FUNCTION_BLOCK "LAF_GetSinaEpos"
TITLE = LAF_GetSinaEpos
{ S7_Optimized_Access := 'TRUE' ; Published := 'TRUE' }
AUTHOR : 'Siemens Digital Industries'
FAMILY : LAF
VERSION : 1.2
//This block reads EPOS positioning status information as well as setpoint and actual values from a SINAMICS drive via acyclic communication depending on the configured type of SINAMICS and the selected drive object index in the HMI by the operator.
   VAR_INPUT
      enable { S7_PredefinedAssignment := 'TRUE'} : Bool := TRUE;   // FALSE = Disables functionality of FB from user program (optional), FB is normally enabled via HMI ('moduleInterface.hmi.sinaEposScreenActive' = TRUE)
   END_VAR

   VAR_OUTPUT
      valid { ExternalWritable := 'False'} : Bool;   // Valid set of output values available at the FB
      busy { ExternalWritable := 'False'} : Bool;   // FB is not finished and new output values can be expected
      error { ExternalWritable := 'False'} : Bool;   // An error occurred during the execution of the FB, for details see diagnostics output
      status { ExternalWritable := 'False'} : Word := #STATUS_NO_CALL;   // 16#0000 - 16#7FFF: Status of the FB, 16#8000 - 16#FFFF: Error identification
      diagnostics { ExternalWritable := 'False'} : "LAF_typeDiagnostics";   // Diagnostics information of FB
      statusWriteRecord { ExternalAccessible := 'False'; ExternalVisible := 'False'; ExternalWritable := 'False'} : DWord;   // Status output of WRREC
      statusReadRecord { ExternalAccessible := 'False'; ExternalVisible := 'False'; ExternalWritable := 'False'} : DWord;   // Status output of RDREC
   END_VAR

   VAR_IN_OUT
      configuration { S7_PredefinedAssignment := 'DriveDiagConfig.driveObjects'} : Array[*] of "LAF_typeDriveDiagConfig";
      moduleInterface { S7_PredefinedAssignment := 'DriveDiagInterfaceHmi.diagStatus'} : "LAF_typeDriveDiagInterfaceHmi";
   END_VAR

   VAR
      statInternal { ExternalAccessible := 'False'; ExternalVisible := 'False'; ExternalWritable := 'False'} : Struct   // Static structure for internal tags
         enablePrevious { ExternalAccessible := 'False'; ExternalVisible := 'False'; ExternalWritable := 'False'} : Bool;   // Previous value of 'enable' input for edge detection
         valid { ExternalAccessible := 'False'; ExternalVisible := 'False'; ExternalWritable := 'False'} : Bool;   // Value for output 'valid'
         busy { ExternalAccessible := 'False'; ExternalVisible := 'False'; ExternalWritable := 'False'} : Bool;   // Value for output 'busy'
         error { ExternalAccessible := 'False'; ExternalVisible := 'False'; ExternalWritable := 'False'} : Bool;   // Value for output 'error'
         errorUserCleared { ExternalAccessible := 'False'; ExternalVisible := 'False'; ExternalWritable := 'False'} : Bool;   // Error occurred that can only be solved by user; rising edge at enable input necessary
         errorAutoCleared { ExternalAccessible := 'False'; ExternalVisible := 'False'; ExternalWritable := 'False'} : Bool;   // Error occurred that can be acknowledged by FB
         disablingCompleted { ExternalAccessible := 'False'; ExternalVisible := 'False'; ExternalWritable := 'False'} : Bool;   // TRUE: Disabling has been completed
         diagnostics { ExternalAccessible := 'False'; ExternalVisible := 'False'; ExternalWritable := 'False'; S7_SetPoint := 'False'} : "LAF_typeDiagnostics" := (#STATUS_NO_CALL, (), ());
         emptyDiagnostics { ExternalAccessible := 'False'; ExternalVisible := 'False'; ExternalWritable := 'False'; S7_SetPoint := 'False'} : "LAF_typeDiagnostics" := (#STATUS_NO_CALL, (), ());   // Empty diagnostics information (for initialization purposes only)
      END_STRUCT;
      statMainState { ExternalAccessible := 'False'; ExternalVisible := 'False'; ExternalWritable := 'False'} : DInt := #FB_STATE_NO_PROCESSING;   // State in the state machine of the FB
      statArrayMin { ExternalAccessible := 'False'; ExternalVisible := 'False'; ExternalWritable := 'False'} : DInt;   // Lower bound of configuration array
      statArrayMax { ExternalAccessible := 'False'; ExternalVisible := 'False'; ExternalWritable := 'False'} : DInt;   // Upper bound of configuration array
      instWriteRecord {InstructionName := 'WRREC'; LibVersion := '1.1'; ExternalAccessible := 'False'; ExternalVisible := 'False'; ExternalWritable := 'False'; S7_SetPoint := 'False'} : WRREC;   // Instance of WRREC
      instReadRecord {InstructionName := 'RDREC'; LibVersion := '1.0'; ExternalAccessible := 'False'; ExternalVisible := 'False'; ExternalWritable := 'False'; S7_SetPoint := 'False'} : RDREC;   // Instance of RDREC
      statWriteReq { ExternalAccessible := 'False'; ExternalVisible := 'False'; ExternalWritable := 'False'} : Struct   // Data of write record according to parameter request
         header { ExternalAccessible := 'False'; ExternalVisible := 'False'; ExternalWritable := 'False'} : Struct   // Request header
            reqRef { ExternalAccessible := 'False'; ExternalVisible := 'False'; ExternalWritable := 'False'} : Byte;   // Unique identification of the request/response pair for the IO controller. The IO device mirrors the request reference in its response
            reqID { ExternalAccessible := 'False'; ExternalVisible := 'False'; ExternalWritable := 'False'} : Byte;   // Specifies the type of request (0x01=read, 0x02=write)
            axis { ExternalAccessible := 'False'; ExternalVisible := 'False'; ExternalWritable := 'False'} : Byte := 16#01;   // Specifies the drive object number for a drive unit with more than one drive object
            noPara { ExternalAccessible := 'False'; ExternalVisible := 'False'; ExternalWritable := 'False'} : Byte := 16#01;   // Number of parameters
         END_STRUCT;
         data { ExternalAccessible := 'False'; ExternalVisible := 'False'; ExternalWritable := 'False'} : Array[0..#DATA_ARRY_MAX] of Byte;   // Request data
      END_STRUCT;
      statReadReq { ExternalAccessible := 'False'; ExternalVisible := 'False'; ExternalWritable := 'False'} : Struct   // Data of read record according to parameter response
         header { ExternalAccessible := 'False'; ExternalVisible := 'False'; ExternalWritable := 'False'} : Struct   // Request header
            reqRef { ExternalAccessible := 'False'; ExternalVisible := 'False'; ExternalWritable := 'False'} : Byte;   // Mirrowed request reference in response of the IO device.
            reqID { ExternalAccessible := 'False'; ExternalVisible := 'False'; ExternalWritable := 'False'} : Byte;   // Mirrowed request identifier. Specifies if request execution was positive or negative (0x01=read+, 0x02=write+, 0x81=read-, 0x82=write-)
            axis { ExternalAccessible := 'False'; ExternalVisible := 'False'; ExternalWritable := 'False'} : Byte := 16#01;   // Specifies the drive object number for a drive unit with more than one drive object
            noPara { ExternalAccessible := 'False'; ExternalVisible := 'False'; ExternalWritable := 'False'} : Byte := 16#01;   // Number of parameters
         END_STRUCT;
         data { ExternalAccessible := 'False'; ExternalVisible := 'False'; ExternalWritable := 'False'} : Array[0..#DATA_ARRY_MAX] of Byte;   // Request data
      END_STRUCT;
      instActTimer {InstructionName := 'IEC_TIMER'; LibVersion := '1.0'; ExternalAccessible := 'False'; ExternalVisible := 'False'; ExternalWritable := 'False'; S7_SetPoint := 'False'} : IEC_TIMER;   // Instance of actual timer for
      instReqTimer {InstructionName := 'IEC_TIMER'; LibVersion := '1.0'; ExternalAccessible := 'False'; ExternalVisible := 'False'; ExternalWritable := 'False'; S7_SetPoint := 'False'} : IEC_TIMER;   // Instance of request timer to retrigger write request
      statDataTransRun { ExternalAccessible := 'False'; ExternalVisible := 'False'; ExternalWritable := 'False'} : Bool;   // Data transfer is running
      statWriteReqSet { ExternalAccessible := 'False'; ExternalVisible := 'False'; ExternalWritable := 'False'} : Bool;   // Parameter for write request set
      statActTimerIn { ExternalAccessible := 'False'; ExternalVisible := 'False'; ExternalWritable := 'False'} : Bool;   // Actual timer start input
      statPrevTimeValue { ExternalAccessible := 'False'; ExternalVisible := 'False'; ExternalWritable := 'False'} : Time;   // Timer value of last trigger
      statActTimerValueAct { ExternalAccessible := 'False'; ExternalVisible := 'False'; ExternalWritable := 'False'} : Time;   // Current timer value of actual timer
      statActTimerValueReq { ExternalAccessible := 'False'; ExternalVisible := 'False'; ExternalWritable := 'False'} : Time;   // Current timer value of request timer
      statPrevDriveIndex { ExternalAccessible := 'False'; ExternalVisible := 'False'; ExternalWritable := 'False'} : DInt;   // Previous drive index
   END_VAR

   VAR_TEMP
      tempEnable : Bool;   // Temporary value for input 'enable'
      tempReferenceDesignator : WString[128];   // Temporary value for inout 'referenceDesignator'
      tempDriveIndex : DInt;   // Temporary value for inout 'driveIndex'
      tempSinaType : UInt;   // Temporary value for inout 'sinaType'
      tempSinaHwID : HW_IO;   // Temporary value for inout 'sinaHwID'
      tempDriveObjectNo : USInt;   // Temporary value for inout 'driveObjectNo'
      tempActTimerOut : Bool;   // Actual timer output
      tempReadReqTimerOut : Bool;   // Request timer output
      tempValueWord : Word;   // Temporary value for 16bit
      tempValueDword : DWord;   // Temporary value for 32bit
   END_VAR

   VAR CONSTANT
      FB_STATE_NO_PROCESSING : DInt := 0;   // FB state: No processing
      FB_STATE_ENABLING : DInt := 10;   // FB state: Enabling
      FB_STATE_PROCESSING : DInt := 50;   // FB state: Processing
      FB_STATE_DISABLING : DInt := 90;   // FB state: Disabling
      STATUS_NO_CALL : Word := 16#7000;   // No job being currently processed
      STATUS_FIRST_CALL : Word := 16#7001;   // First call after incoming new job (rising edge 'enable')
      STATUS_SUBSEQUENT_CALL : Word := 16#7002;   // Subsequent call during active processing without further details
      STATUS_WARN_ARRY_MIN : Word := 16#7003;   // Active processing with index assigned to lower bound of configuration arry
      STATUS_WARN_ARRY_MAX : Word := 16#7004;   // Active processing with index assigned to upper bound of configuration arry
      STAUTS_WARN_NO_SINAMICS : Word := 16#7005;   // Selected SINAMICS type in configuration not supported. Active processing with SINAMICS type assigned to no type.
      STAUTS_WARN_DO_SINGLE_AXIS : Word := 16#7006;   // Active processing with drive object number assigned to single-axis
      SUB_STATUS_NO_ERROR : Word := 16#0000;   // NO error occurred in sub function call
      ERR_UNDEFINED_STATE : Word := 16#8600;   // Error: due to an undefined state in state machine
      DIM_ARRAY_CONFIG : UDInt := 1;   // Dimension of the configuration array
      DRV_INDEX_INIT : DInt := -1;   // Initial value for drive index
      DRV_DO_SINGLE_AXIS : USInt := 1;   // Drive object number for single-axis
      DATA_ARRY_MAX : UInt := 235;   // Maximum size in bytes for request/response data
      DPV1_INDEX_DB47 : DInt := 47;   // DPV1 services PROFIBUS/PROFINET: Data block 47
      DPV1_LENGH_DATA : UInt := 240;   // DPV1 services PROFIBUS/PROFINET: Maximum length in bytes of the data record information
      TYPE_OF_SINA_NO_TYPE : UInt := 0;   // Type of SINAMICS not specified
      TYPE_OF_SINA_G120 : UInt := 114;   // Type of SINAMICS is G120
      TYPE_OF_SINA_G220 : UInt := 214;   // Type of SINAMICS is G220
      TYPE_OF_SINA_S120 : UInt := 124;   // Type of SINAMICS is S120
      TYPE_OF_SINA_S120_EPOS : UInt := 125;   // Type of SINAMICS is S120 with EPOS
      TYPE_OF_SINA_S200 : UInt := 220;   // Type of SINAMICS is S200
      TYPE_OF_SINA_S200_EPOS : UInt := 221;   // Type of SINAMICS is S200 with EPOS
      TYPE_OF_SINA_S210 : UInt := 222;   // Type of SINAMICS is S210
      TYPE_OF_SINA_S210_EPOS : UInt := 223;   // Type of SINAMICS is S210 with EPOS
      TYPE_OF_SINA_S220 : UInt := 224;   // Type of SINAMICS is S220
      TYPE_OF_SINA_S220_EPOS : UInt := 225;   // Type of SINAMICS is S220 with EPOS
      REQ_ID_READ : Byte := 16#01;   // Specifies read request for WRREC
      REQ_ID_WRITE : Byte := 16#02;   // Specifies write request for WRREC
      REQ_REF_G120 : Byte := 32;   // Response ID of response request of G120
      REQ_REF_G220 : Byte := 132;   // Response ID of response request of G220
      REQ_REF_S120 : Byte := 62;   // Response ID of response request of S120
      REQ_REF_S200 : Byte := 142;   // Response ID of response request of S200
      REQ_REF_S210 : Byte := 152;   // Response ID of response request of S210
      REQ_REF_S220 : Byte := 162;   // Response ID of response request of S220
   END_VAR


BEGIN
	REGION BLOCK INFO HEADER
	    //===============================================================================
	    // Siemens AG / (c)Copyright 2024
	    //-------------------------------------------------------------------------------
	    // Title:            LAF_GetSinaEpos
	    // Comment/Function: This block reads EPOS positioning status information as well
	    //                   as setpoint and actual values from a SINAMICS drive via
	    //                   acyclic communication depending on the configured type of
	    //                   SINAMICS and the selected drive object index in the HMI
	    //                   by the operator.
	    // Library/Family:   Automation Framework / Drive Diagnostic
	    // Author:           Siemens Digital Industries
	    // Tested with:      S7-PLCSIM Advanced 6.0
	    // Engineering:      TIA Portal V19
	    // Restrictions:     -
	    // Requirements:     -
	    //-------------------------------------------------------------------------------
	    // Change log table:
	    // Version  | Date       | Expert in charge        | Changes applied
	    //----------|------------|-------------------------|-----------------------------
	    // 01.00.00 | 15.12.2023 | SIMATIC Systems Support | First released version
	    // 01.01.00 | 30.06.2024 | SIMATIC Systems Support | UDTs updated, Enable/Disable
	    // 01.02.00 | 30.09.2024 | SIMATIC Systems Support | Block information properties updated
	    //===============================================================================
	END_REGION BLOCK INFO HEADER

	REGION DESCRIPTION
	(/*
	This block reads EPOS positioning status information as well as setpoint and actual values
	via PROFIBUS/PROFINET from a SINAMICS drive, by using acyclic communication with
	"Write data record" and "Read data record" services via the PROFIdrive parameter channel
	with data block 47 and the WRREC and RDREC system blocks.
	At runtime, this block is enabled when the SINAMCIS EPOS status diagnostic screen is shown
	in the HMI. Based on the selected drive object (index) in the HMI by the operator, the EPOS status
	is read out from the SINAMICS and transmitted to the HMI.
	The shown EPOS status in the HMI depends on the type of SINAMICS(S120_EPOS, S200_EPOS, S210_EPOS).
	Therefore the type of SINAMICS must be specified in the configuration DB. In addition, the
	hardware identifier (HW_IO) and the number of the drive object (DO) must be configured too.
	*/)
	END_REGION

	REGION INPUTS
	    // Work with temporary values / create process image
	    #tempEnable := #enable AND #moduleInterface.hmi.sinaEposScreenActive;
	    #tempDriveIndex := #moduleInterface.hmi.driveIndex;
	END_REGION INPUTS

	REGION ENABLING/DISABLING
	    IF (#tempEnable = TRUE) AND (#statInternal.diagnostics.status = #STATUS_NO_CALL) THEN // Enable FB
	        // First call; initialize FB
	        #statInternal.valid := TRUE;
	        #statInternal.busy := TRUE;
	        #statInternal.error := FALSE;
	        #statInternal.errorUserCleared := FALSE;
	        #statInternal.errorAutoCleared := FALSE;
	        #statInternal.disablingCompleted := FALSE;
	        #statInternal.diagnostics := #statInternal.emptyDiagnostics;
	        #diagnostics := #statInternal.emptyDiagnostics;
	        #statInternal.diagnostics.status := #STATUS_FIRST_CALL;
	        // State machine - start processing
	        #statMainState := #FB_STATE_ENABLING;
	        // Initialize diagnostic data
	        #statusWriteRecord := W#16#00;
	        #statusReadRecord := W#16#00;
	        #statPrevDriveIndex := #DRV_INDEX_INIT;
	        #moduleInterface.sina.sinaType := 0;
	        #moduleInterface.sina.statusWord := W#16#0;
	        #moduleInterface.sina.eposStatusWord1 := W#16#0;
	        #moduleInterface.sina.eposStatusWord2 := W#16#0;
	        #moduleInterface.sina.operatingDisplay := 0;
	        #moduleInterface.sina.override := 0.0;
	        #moduleInterface.sina.posSetValue := 0.0;
	        #moduleInterface.sina.posActValue := 0.0;
	        #moduleInterface.sina.velSetValue := 0.0;
	        #moduleInterface.sina.velActValue := 0.0;
	        #moduleInterface.sina.lengthUnit := 0;
	        #moduleInterface.sina.velocityUnit := 0;
	        #moduleInterface.sina.residualDistance := 0.0;
	        #moduleInterface.sina.followingError := 0.0;
	        #moduleInterface.sina.posControlWord := W#16#0;
	        #moduleInterface.sina.posStatusWord := W#16#0;
	        #moduleInterface.sina.blockSelected := 0;
	        #moduleInterface.sina.blockActive := 0;
	        #moduleInterface.sina.mdiPosSetValue := 0.0;

	    ELSIF (#tempEnable = FALSE) AND (#statInternal.enablePrevious = TRUE) THEN // Disable FB
	        #statMainState := #FB_STATE_DISABLING;

	    ELSIF (#statInternal.diagnostics.status = #STATUS_FIRST_CALL) THEN // Set status identifier of subsequent call
	        #statInternal.diagnostics.status := #STATUS_SUBSEQUENT_CALL;
	    END_IF;

	    // Edge detection 'tempEnable'
	    #statInternal.enablePrevious := #tempEnable;
	END_REGION ENABLING/DISABLING

	IF (#statInternal.diagnostics.status = #STATUS_NO_CALL) THEN // Nothing to do -> End here to reduce "system load"
	    RETURN;
	END_IF;

	REGION STATE MACHINE
	    CASE #statMainState OF // State machine of FB
	        #FB_STATE_NO_PROCESSING:
	            REGION No Processing
	                ; // No processing active (Note: this state must always be present and left empty)
	            END_REGION No Processing

	        #FB_STATE_ENABLING: // Enabling active
	            REGION Enabling
	                // Initialize boundaries of configuration array
	                #statArrayMin := LOWER_BOUND(ARR := #configuration, DIM := #DIM_ARRAY_CONFIG);
	                #statArrayMax := UPPER_BOUND(ARR := #configuration, DIM := #DIM_ARRAY_CONFIG);
	                // Continue processing with next state
	                #statMainState := #FB_STATE_PROCESSING;
	            END_REGION Enabling

	        #FB_STATE_PROCESSING: // Processing active
	            REGION Processing
	                // When index is off boundaries, index is assigned to violated bound and active processing with warning
	                IF (#tempDriveIndex < #statArrayMin) THEN
	                    #tempDriveIndex := #statArrayMin;
	                    #statInternal.diagnostics.status := #STATUS_WARN_ARRY_MIN;
	                    #statInternal.diagnostics.subfunctionStatus := #SUB_STATUS_NO_ERROR;
	                    #statInternal.diagnostics.stateNumber := #statMainState;
	                ELSIF (#tempDriveIndex > #statArrayMax) THEN
	                    #tempDriveIndex := #statArrayMax;
	                    #statInternal.diagnostics.status := #STATUS_WARN_ARRY_MAX;
	                    #statInternal.diagnostics.subfunctionStatus := #SUB_STATUS_NO_ERROR;
	                    #statInternal.diagnostics.stateNumber := #statMainState;
	                ELSE
	                    #statInternal.diagnostics.status := #STATUS_SUBSEQUENT_CALL;
	                    #statInternal.diagnostics.subfunctionStatus := #SUB_STATUS_NO_ERROR;
	                    #statInternal.diagnostics.stateNumber := #statMainState;
	                END_IF;

	                // Work with temporary values
	                #tempReferenceDesignator := #configuration[#tempDriveIndex].referenceDesignator;
	                #tempSinaType := #configuration[#tempDriveIndex].sinaType;
	                #tempSinaHwID := #configuration[#tempDriveIndex].sinaHwID;
	                #tempDriveObjectNo := #configuration[#tempDriveIndex].sinaDriveObjectNo;

	                // When SINAMICS type is not supported, type is assigned to no type
	                IF (#tempSinaType <> #TYPE_OF_SINA_G120) AND
	                    (#tempSinaType <> #TYPE_OF_SINA_S120) AND
	                    (#tempSinaType <> #TYPE_OF_SINA_S120_EPOS) AND
	                    (#tempSinaType <> #TYPE_OF_SINA_S200) AND
	                    (#tempSinaType <> #TYPE_OF_SINA_S200_EPOS) AND
	                    (#tempSinaType <> #TYPE_OF_SINA_S210) AND
	                    (#tempSinaType <> #TYPE_OF_SINA_S210_EPOS)
	                THEN
	                    #tempSinaType := #TYPE_OF_SINA_NO_TYPE;
	                    #statInternal.diagnostics.status := #STAUTS_WARN_NO_SINAMICS;
	                    #statInternal.diagnostics.subfunctionStatus := #SUB_STATUS_NO_ERROR;
	                    #statInternal.diagnostics.stateNumber := #statMainState;
	                END_IF;

	                // Check drive object number
	                IF (#tempDriveObjectNo < #DRV_DO_SINGLE_AXIS) THEN
	                    #tempDriveObjectNo := #DRV_DO_SINGLE_AXIS;
	                    #statInternal.diagnostics.status := #STAUTS_WARN_DO_SINGLE_AXIS;
	                    #statInternal.diagnostics.subfunctionStatus := #SUB_STATUS_NO_ERROR;
	                    #statInternal.diagnostics.stateNumber := #statMainState;
	                END_IF;

	                // Set SINAMICS type
	                #moduleInterface.sina.sinaType := #tempSinaType;

	                // Actual timer for communication with drive
	                #instActTimer.TON(IN := #statActTimerIn,
	                                  PT := T#596h,
	                                  Q => #tempActTimerOut,
	                                  ET => #statActTimerValueAct);
	                IF NOT #tempActTimerOut THEN
	                    #statActTimerIn := true;
	                ELSE
	                    #statActTimerIn := FALSE;
	                    #statPrevTimeValue := T#0s;
	                END_IF;

	                // Initialize dataö
	                IF #tempDriveIndex <> #statPrevDriveIndex THEN
	                    // Write request
	                    #statWriteReq.header.reqRef := B#16#00;
	                    #statWriteReq.header.reqID := B#16#00;
	                    #statWriteReq.header.axis := B#16#01;
	                    #statWriteReq.header.noPara := B#16#00;
	                    FILL_BLK(IN := B#16#00,
	                             COUNT := #DATA_ARRY_MAX + 1,
	                             OUT => #statWriteReq.data[0]);
	                    #statWriteReqSet := FALSE;
	                    // Read request
	                    #statReadReq.header.reqRef := B#16#00;
	                    #statReadReq.header.reqID := B#16#00;
	                    #statReadReq.header.axis := B#16#01;
	                    #statReadReq.header.noPara := B#16#00;
	                    FILL_BLK(IN := B#16#00,
	                             COUNT := #DATA_ARRY_MAX + 1,
	                             OUT => #statReadReq.data[0]);
	                    #statDataTransRun := FALSE;
	                    // Diagnostic data
	                    #statusWriteRecord := W#16#00;
	                    #statusReadRecord := W#16#00;
	                    #moduleInterface.sina.sinaType := 0;
	                    #moduleInterface.sina.statusWord := W#16#0;
	                    #moduleInterface.sina.eposStatusWord1 := W#16#0;
	                    #moduleInterface.sina.eposStatusWord2 := W#16#0;
	                    #moduleInterface.sina.operatingDisplay := 0;
	                    #moduleInterface.sina.override := 0.0;
	                    #moduleInterface.sina.posSetValue := 0.0;
	                    #moduleInterface.sina.posActValue := 0.0;
	                    #moduleInterface.sina.velSetValue := 0.0;
	                    #moduleInterface.sina.velActValue := 0.0;
	                    #moduleInterface.sina.lengthUnit := 0;
	                    #moduleInterface.sina.velocityUnit := 0;
	                    #moduleInterface.sina.residualDistance := 0.0;
	                    #moduleInterface.sina.followingError := 0.0;
	                    #moduleInterface.sina.posControlWord := W#16#0;
	                    #moduleInterface.sina.posStatusWord := W#16#0;
	                    #moduleInterface.sina.blockSelected := 0;
	                    #moduleInterface.sina.blockActive := 0;
	                    #moduleInterface.sina.mdiPosSetValue := 0.0;
	                    // Memorize previous selected drive object
	                    #statPrevDriveIndex := #moduleInterface.hmi.driveIndex;
	                END_IF;

	                REGION Write request
	                    CASE #tempSinaType OF
	                        #TYPE_OF_SINA_S120_EPOS:
	                            REGION S120
	                                // Order header
	                                #statWriteReq.header.reqRef := #REQ_REF_S120; // Order reference
	                                #statWriteReq.header.reqID := #REQ_ID_READ; // Reading order
	                                #statWriteReq.header.axis := USINT_TO_BYTE(#tempDriveObjectNo); // Drive object number
	                                #statWriteReq.header.noPara := 14; //Number of parameters
	                                // 1. Drive parameter r2683 (EPOS status word 1) in hex 0x0A7B
	                                #statWriteReq.data[0] := B#16#10; // Read parameter values
	                                #statWriteReq.data[1] := B#16#01; // Number of elements
	                                #statWriteReq.data[2] := B#16#0A; // Parameter number r2683 (EPOS status word 1) high byte
	                                #statWriteReq.data[3] := B#16#7B; // Parameter number r2683 (EPOS status word 1) low byte
	                                #statWriteReq.data[4] := B#16#00; // Subindex
	                                #statWriteReq.data[5] := B#16#00; // Subindex
	                                // 2. Drive parameter r2684 (EPOS status word 2) in hex 0x0A7C
	                                #statWriteReq.data[6] := B#16#10; // Read parameter values
	                                #statWriteReq.data[7] := B#16#01; // Number of elements
	                                #statWriteReq.data[8] := B#16#0A; // Parameter number r2684 (EPOS status word 2) high byte
	                                #statWriteReq.data[9] := B#16#7C; // Parameter number r2684 (EPOS status word 2) low byte
	                                #statWriteReq.data[10] := B#16#00; // Subindex
	                                #statWriteReq.data[11] := B#16#00; // Subindex
	                                // 3. Drive parameter r0002 (Operating display) in hex 0x0002
	                                #statWriteReq.data[12] := B#16#10; // Read parameter values
	                                #statWriteReq.data[13] := B#16#01; // Number of elements
	                                #statWriteReq.data[14] := B#16#00; // Parameter number r0002 (Operating display) high byte
	                                #statWriteReq.data[15] := B#16#02; // Parameter number r0002 (Operating display) low byte
	                                #statWriteReq.data[16] := B#16#00; // Subindex
	                                #statWriteReq.data[17] := B#16#00; // Subindex
	                                // 4. Drive parameter r2681 (Override) in hex 0A79
	                                #statWriteReq.data[18] := B#16#10; // Read parameter values
	                                #statWriteReq.data[19] := B#16#01; // Number of elements
	                                #statWriteReq.data[20] := B#16#0A; // Parameter number r2681 (Override) high byte
	                                #statWriteReq.data[21] := B#16#79; // Parameter number r2681 (Override) low byte
	                                #statWriteReq.data[22] := B#16#00; // Subindex
	                                #statWriteReq.data[23] := B#16#00; // Subindex
	                                // 5. Drive parameter r2666 (setpoint velocity) in hex 0x0A6A
	                                #statWriteReq.data[24] := B#16#10; // Read parameter values
	                                #statWriteReq.data[25] := B#16#01; // Number of elements
	                                #statWriteReq.data[26] := B#16#0A; // Parameter number r2666 (setpoint velocity) high byte
	                                #statWriteReq.data[27] := B#16#6A; // Parameter number r2666 (setpoint velocity) low byte
	                                #statWriteReq.data[28] := B#16#00; // Subindex
	                                #statWriteReq.data[29] := B#16#00; // Subindex
	                                // 6. Drive parameter r2522[0] (actual velocity) in hex 0x09DA
	                                #statWriteReq.data[30] := B#16#10; // Read parameter values
	                                #statWriteReq.data[31] := B#16#01; // Number of elements
	                                #statWriteReq.data[32] := B#16#09; // Parameter number r2522[0] (actual velocity) high byte
	                                #statWriteReq.data[33] := B#16#DA; // Parameter number r2522[0] (actual velocity) low byte
	                                #statWriteReq.data[34] := B#16#00; // Subindex
	                                #statWriteReq.data[35] := B#16#00; // Subindex
	                                // 7. Drive parameter r2665 (setpoint position) in hex 0x0A69
	                                #statWriteReq.data[36] := B#16#10; // Read parameter values
	                                #statWriteReq.data[37] := B#16#01; // Number of elements
	                                #statWriteReq.data[38] := B#16#0A; // Parameter number r2665 (setpoint position) high byte
	                                #statWriteReq.data[39] := B#16#69; // Parameter number r2665 (setpoint position) low byte
	                                #statWriteReq.data[40] := B#16#00; // Subindex
	                                #statWriteReq.data[41] := B#16#00; // Subindex
	                                // 8. Drive parameter r2521[0] (actual position) in hex 0x09D9
	                                #statWriteReq.data[42] := B#16#10; // Read parameter values
	                                #statWriteReq.data[43] := B#16#01; // Number of elements
	                                #statWriteReq.data[44] := B#16#09; // Parameter number r2521[0] (actual position) high byte
	                                #statWriteReq.data[45] := B#16#D9; // Parameter number r2521[0] (actual position) low byte
	                                #statWriteReq.data[46] := B#16#00; // Subindex
	                                #statWriteReq.data[47] := B#16#00; // Subindex
	                                // 9. Drive parameter r2682 (residual distance) in hex 0x0A7A
	                                #statWriteReq.data[48] := B#16#10; // Read parameter values
	                                #statWriteReq.data[49] := B#16#01; // Number of elements
	                                #statWriteReq.data[50] := B#16#0A; // Parameter number r2682 (residual distance) high byte
	                                #statWriteReq.data[51] := B#16#7A; // Parameter number r2682 (residual distance) low byte
	                                #statWriteReq.data[52] := B#16#00; // Subindex
	                                #statWriteReq.data[53] := B#16#00; // Subindex
	                                // 10. Drive parameter r2565 (following error) in hex 0x0A05
	                                #statWriteReq.data[54] := B#16#10; // Read parameter values
	                                #statWriteReq.data[55] := B#16#01; // Number of elements
	                                #statWriteReq.data[56] := B#16#0A; // Parameter number r2565 (following error) high byte
	                                #statWriteReq.data[57] := B#16#05; // Parameter number r2565 (following error) low byte
	                                #statWriteReq.data[58] := B#16#00; // Subindex
	                                #statWriteReq.data[59] := B#16#00; // Subindex
	                                // 11. Drive parameter r2091 (positioning control word) in hex 0x082B
	                                #statWriteReq.data[60] := B#16#10; // Read parameter values
	                                #statWriteReq.data[61] := B#16#01; // Number of elements
	                                #statWriteReq.data[62] := B#16#08; // Parameter number r2091 (positioning control word) high byte
	                                #statWriteReq.data[63] := B#16#2B; // Parameter number r2091 (positioning control word) low byte
	                                #statWriteReq.data[64] := B#16#00; // Subindex
	                                #statWriteReq.data[65] := B#16#00; // Subindex
	                                // 12. Drive parameter r2053[1] (positioning status word) in hex 0x0805
	                                #statWriteReq.data[66] := B#16#10; // Read parameter values
	                                #statWriteReq.data[67] := B#16#01; // Number of elements
	                                #statWriteReq.data[68] := B#16#08; // Parameter number r2053[1] (positioning status word) high byte
	                                #statWriteReq.data[69] := B#16#05; // Parameter number r2053[1] (positioning status word) low byte
	                                #statWriteReq.data[70] := B#16#00; // Subindex
	                                #statWriteReq.data[71] := B#16#01; // Subindex
	                                // 13. Drive parameter r2060[5] (MDI setpoint position) in hex 0x080C
	                                #statWriteReq.data[72] := B#16#10; // Read parameter values
	                                #statWriteReq.data[73] := B#16#01; // Number of elements
	                                #statWriteReq.data[74] := B#16#08; // Parameter number r2060[5] (MDI setpoint position) high byte
	                                #statWriteReq.data[75] := B#16#0C; // Parameter number r2060[5] (MDI setpoint position) low byte
	                                #statWriteReq.data[76] := B#16#00; // Subindex
	                                #statWriteReq.data[77] := B#16#05; // Subindex
	                                // 14. Drive parameter r2089[0] (#status word) in hex 0x0829
	                                #statWriteReq.data[78] := B#16#10; // Read parameter values
	                                #statWriteReq.data[79] := B#16#01; // Number of elements
	                                #statWriteReq.data[80] := B#16#08; // Parameter number r2089[0] (status word) high byte
	                                #statWriteReq.data[81] := B#16#29; // Parameter number r2089[0] (status word) low byte
	                                #statWriteReq.data[82] := B#16#00; // Subindex
	                                #statWriteReq.data[83] := B#16#00; // Subindex
	                                // Start request
	                                #statWriteReqSet := TRUE;
	                                #statDataTransRun := TRUE;
	                            END_REGION S120

	                        #TYPE_OF_SINA_S200_EPOS:
	                            REGION S200
	                                // Order header
	                                #statWriteReq.header.reqRef := #REQ_REF_S200; // Order reference
	                                #statWriteReq.header.reqID := #REQ_ID_READ; // Reading order
	                                #statWriteReq.header.axis := USINT_TO_BYTE(#tempDriveObjectNo); // Drive object number
	                                #statWriteReq.header.noPara := 16; //Number of parameters
	                                // 1. Drive parameter r2683 (EPOS status word 1) in hex 0x0A7B
	                                #statWriteReq.data[0] := B#16#10; // Read parameter values
	                                #statWriteReq.data[1] := B#16#01; // Number of elements
	                                #statWriteReq.data[2] := B#16#0A; // Parameter number r2683 (EPOS status word 1) high byte
	                                #statWriteReq.data[3] := B#16#7B; // Parameter number r2683 (EPOS status word 1) low byte
	                                #statWriteReq.data[4] := B#16#00; // Subindex
	                                #statWriteReq.data[5] := B#16#00; // Subindex
	                                // 2. Drive parameter r2684 (EPOS status word 2) in hex 0x0A7C
	                                #statWriteReq.data[6] := B#16#10; // Read parameter values
	                                #statWriteReq.data[7] := B#16#01; // Number of elements
	                                #statWriteReq.data[8] := B#16#0A; // Parameter number r2684 (EPOS status word 2) high byte
	                                #statWriteReq.data[9] := B#16#7C; // Parameter number r2684 (EPOS status word 2) low byte
	                                #statWriteReq.data[10] := B#16#00; // Subindex
	                                #statWriteReq.data[11] := B#16#00; // Subindex
	                                // 3. Drive parameter r0002 (Operating display) in hex 0x0002
	                                #statWriteReq.data[12] := B#16#10; // Read parameter values
	                                #statWriteReq.data[13] := B#16#01; // Number of elements
	                                #statWriteReq.data[14] := B#16#00; // Parameter number r0002 (Operating display) high byte
	                                #statWriteReq.data[15] := B#16#02; // Parameter number r0002 (Operating display) low byte
	                                #statWriteReq.data[16] := B#16#00; // Subindex
	                                #statWriteReq.data[17] := B#16#00; // Subindex
	                                // 4. Drive parameter c2646 (Override) in hex 0A56
	                                #statWriteReq.data[18] := B#16#10; // Read parameter values
	                                #statWriteReq.data[19] := B#16#01; // Number of elements
	                                #statWriteReq.data[20] := B#16#0A; // Parameter number c2646 (Override) high byte
	                                #statWriteReq.data[21] := B#16#56; // Parameter number c2646 (Override) low byte
	                                #statWriteReq.data[22] := B#16#00; // Subindex
	                                #statWriteReq.data[23] := B#16#00; // Subindex
	                                // 5. Drive parameter r2666 (setpoint velocity) in hex 0x0A6A
	                                #statWriteReq.data[24] := B#16#10; // Read parameter values
	                                #statWriteReq.data[25] := B#16#01; // Number of elements
	                                #statWriteReq.data[26] := B#16#0A; // Parameter number r2666 (setpoint velocity) high byte
	                                #statWriteReq.data[27] := B#16#6A; // Parameter number r2666 (setpoint velocity) low byte
	                                #statWriteReq.data[28] := B#16#00; // Subindex
	                                #statWriteReq.data[29] := B#16#00; // Subindex
	                                // 6. Drive parameter r2522[0] (actual velocity) in hex 0x09DA
	                                #statWriteReq.data[30] := B#16#10; // Read parameter values
	                                #statWriteReq.data[31] := B#16#01; // Number of elements
	                                #statWriteReq.data[32] := B#16#09; // Parameter number r2522[0] (actual velocity) high byte
	                                #statWriteReq.data[33] := B#16#DA; // Parameter number r2522[0] (actual velocity) low byte
	                                #statWriteReq.data[34] := B#16#00; // Subindex
	                                #statWriteReq.data[35] := B#16#00; // Subindex
	                                // 7. Drive parameter r2665 (setpoint position) in hex 0x0A69
	                                #statWriteReq.data[36] := B#16#10; // Read parameter values
	                                #statWriteReq.data[37] := B#16#01; // Number of elements
	                                #statWriteReq.data[38] := B#16#0A; // Parameter number r2665 (setpoint position) high byte
	                                #statWriteReq.data[39] := B#16#69; // Parameter number r2665 (setpoint position) low byte
	                                #statWriteReq.data[40] := B#16#00; // Subindex
	                                #statWriteReq.data[41] := B#16#00; // Subindex
	                                // 8. Drive parameter r2521[0] (actual position) in hex 0x09D9
	                                #statWriteReq.data[42] := B#16#10; // Read parameter values
	                                #statWriteReq.data[43] := B#16#01; // Number of elements
	                                #statWriteReq.data[44] := B#16#09; // Parameter number r2521[0] (actual position) high byte
	                                #statWriteReq.data[45] := B#16#D9; // Parameter number r2521[0] (actual position) low byte
	                                #statWriteReq.data[46] := B#16#00; // Subindex
	                                #statWriteReq.data[47] := B#16#00; // Subindex
	                                // 9. Drive parameter r2496 (length unit) in hex 0x09C0
	                                #statWriteReq.data[48] := B#16#10; // Read parameter values
	                                #statWriteReq.data[49] := B#16#01; // Number of elements
	                                #statWriteReq.data[50] := B#16#09; // Parameter number r2496 (length unit) high byte
	                                #statWriteReq.data[51] := B#16#C0; // Parameter number r2496 (length unit) low byte
	                                #statWriteReq.data[52] := B#16#00; // Subindex
	                                #statWriteReq.data[53] := B#16#00; // Subindex
	                                // 10. Drive parameter r2497 (velocity unit) in hex 0x09C1
	                                #statWriteReq.data[54] := B#16#10; // Read parameter values
	                                #statWriteReq.data[55] := B#16#01; // Number of elements
	                                #statWriteReq.data[56] := B#16#09; // Parameter number r2497 (velocity unit) high byte
	                                #statWriteReq.data[57] := B#16#C1; // Parameter number r2497 (velocity unit) low byte
	                                #statWriteReq.data[58] := B#16#00; // Subindex
	                                #statWriteReq.data[59] := B#16#00; // Subindex
	                                // 11. Drive parameter r2682 (residual distance) in hex 0x0A7A
	                                #statWriteReq.data[60] := B#16#10; // Read parameter values
	                                #statWriteReq.data[61] := B#16#01; // Number of elements
	                                #statWriteReq.data[62] := B#16#0A; // Parameter number r2682 (residual distance) high byte
	                                #statWriteReq.data[63] := B#16#7A; // Parameter number r2682 (residual distance) low byte
	                                #statWriteReq.data[64] := B#16#00; // Subindex
	                                #statWriteReq.data[65] := B#16#00; // Subindex
	                                // 12. Drive parameter r2565 (following error) in hex 0x0A05
	                                #statWriteReq.data[66] := B#16#10; // Read parameter values
	                                #statWriteReq.data[67] := B#16#01; // Number of elements
	                                #statWriteReq.data[68] := B#16#0A; // Parameter number r2565 (following error) high byte
	                                #statWriteReq.data[69] := B#16#05; // Parameter number r2565 (following error) low byte
	                                #statWriteReq.data[70] := B#16#00; // Subindex
	                                #statWriteReq.data[71] := B#16#00; // Subindex
	                                // 13. Drive parameter r2050[1] (positioning control word) in hex 0x0802
	                                #statWriteReq.data[72] := B#16#10; // Read parameter values
	                                #statWriteReq.data[73] := B#16#01; // Number of elements
	                                #statWriteReq.data[74] := B#16#08; // Parameter number r2050[1] (positioning control word) high byte
	                                #statWriteReq.data[75] := B#16#02; // Parameter number r2050[1] (positioning control word) low byte
	                                #statWriteReq.data[76] := B#16#00; // Subindex
	                                #statWriteReq.data[77] := B#16#01; // Subindex
	                                // 14. Drive parameter c2053[1] (positioning status word) in hex 0x0805
	                                #statWriteReq.data[78] := B#16#10; // Read parameter values
	                                #statWriteReq.data[79] := B#16#01; // Number of elements
	                                #statWriteReq.data[80] := B#16#08; // Parameter number c2053[1] (positioning status word) high byte
	                                #statWriteReq.data[81] := B#16#05; // Parameter number c2053[1] (positioning status word) low byte
	                                #statWriteReq.data[82] := B#16#00; // Subindex
	                                #statWriteReq.data[83] := B#16#01; // Subindex
	                                // 15. Drive parameter c2642 (MDI setpoint position) in hex 0x0A52
	                                #statWriteReq.data[84] := B#16#10; // Read parameter values
	                                #statWriteReq.data[85] := B#16#01; // Number of elements
	                                #statWriteReq.data[86] := B#16#0A; // Parameter number c2642 (MDI setpoint position) high byte
	                                #statWriteReq.data[87] := B#16#52; // Parameter number c2642 (MDI setpoint position) low byte
	                                #statWriteReq.data[88] := B#16#00; // Subindex
	                                #statWriteReq.data[89] := B#16#00; // Subindex
	                                // 16. Drive parameter c2053[0] (status word) in hex 0x0805
	                                #statWriteReq.data[90] := B#16#10; // Read parameter values
	                                #statWriteReq.data[91] := B#16#01; // Number of elements
	                                #statWriteReq.data[92] := B#16#08; // Parameter number c2053[0] (status word) high byte
	                                #statWriteReq.data[93] := B#16#05; // Parameter number c2053[0] (status word) low byte
	                                #statWriteReq.data[94] := B#16#00; // Subindex
	                                #statWriteReq.data[95] := B#16#00; // Subindex
	                                // Start request
	                                #statWriteReqSet := TRUE;
	                                #statDataTransRun := TRUE;
	                            END_REGION S200

	                        #TYPE_OF_SINA_S210_EPOS:
	                            REGION S210
	                                // Order header
	                                #statWriteReq.header.reqRef := #REQ_REF_S210; // Order reference
	                                #statWriteReq.header.reqID := #REQ_ID_READ; // Reading order
	                                #statWriteReq.header.axis := USINT_TO_BYTE(#tempDriveObjectNo); // Drive object number
	                                #statWriteReq.header.noPara := 16; //Number of parameters
	                                // 1. Drive parameter r2683 (EPOS status word 1) in hex 0x0A7B
	                                #statWriteReq.data[0] := B#16#10; // Read parameter values
	                                #statWriteReq.data[1] := B#16#01; // Number of elements
	                                #statWriteReq.data[2] := B#16#0A; // Parameter number r2683 (EPOS status word 1) high byte
	                                #statWriteReq.data[3] := B#16#7B; // Parameter number r2683 (EPOS status word 1) low byte
	                                #statWriteReq.data[4] := B#16#00; // Subindex
	                                #statWriteReq.data[5] := B#16#00; // Subindex
	                                // 2. Drive parameter r2684 (EPOS status word 2) in hex 0x0A7C
	                                #statWriteReq.data[6] := B#16#10; // Read parameter values
	                                #statWriteReq.data[7] := B#16#01; // Number of elements
	                                #statWriteReq.data[8] := B#16#0A; // Parameter number r2684 (EPOS status word 2) high byte
	                                #statWriteReq.data[9] := B#16#7C; // Parameter number r2684 (EPOS status word 2) low byte
	                                #statWriteReq.data[10] := B#16#00; // Subindex
	                                #statWriteReq.data[11] := B#16#00; // Subindex
	                                // 3. Drive parameter r0002 (Operating display) in hex 0x0002
	                                #statWriteReq.data[12] := B#16#10; // Read parameter values
	                                #statWriteReq.data[13] := B#16#01; // Number of elements
	                                #statWriteReq.data[14] := B#16#00; // Parameter number r0002 (Operating display) high byte
	                                #statWriteReq.data[15] := B#16#02; // Parameter number r0002 (Operating display) low byte
	                                #statWriteReq.data[16] := B#16#00; // Subindex
	                                #statWriteReq.data[17] := B#16#00; // Subindex
	                                // 4. Drive parameter c2646 (Override) in hex 0A56
	                                #statWriteReq.data[18] := B#16#10; // Read parameter values
	                                #statWriteReq.data[19] := B#16#01; // Number of elements
	                                #statWriteReq.data[20] := B#16#0A; // Parameter number c2646 (Override) high byte
	                                #statWriteReq.data[21] := B#16#56; // Parameter number c2646 (Override) low byte
	                                #statWriteReq.data[22] := B#16#00; // Subindex
	                                #statWriteReq.data[23] := B#16#00; // Subindex
	                                // 5. Drive parameter r2666 (setpoint velocity) in hex 0x0A6A
	                                #statWriteReq.data[24] := B#16#10; // Read parameter values
	                                #statWriteReq.data[25] := B#16#01; // Number of elements
	                                #statWriteReq.data[26] := B#16#0A; // Parameter number r2666 (setpoint velocity) high byte
	                                #statWriteReq.data[27] := B#16#6A; // Parameter number r2666 (setpoint velocity) low byte
	                                #statWriteReq.data[28] := B#16#00; // Subindex
	                                #statWriteReq.data[29] := B#16#00; // Subindex
	                                // 6. Drive parameter r2522[0] (actual velocity) in hex 0x09DA
	                                #statWriteReq.data[30] := B#16#10; // Read parameter values
	                                #statWriteReq.data[31] := B#16#01; // Number of elements
	                                #statWriteReq.data[32] := B#16#09; // Parameter number r2522[0] (actual velocity) high byte
	                                #statWriteReq.data[33] := B#16#DA; // Parameter number r2522[0] (actual velocity) low byte
	                                #statWriteReq.data[34] := B#16#00; // Subindex
	                                #statWriteReq.data[35] := B#16#00; // Subindex
	                                // 7. Drive parameter r2665 (setpoint position) in hex 0x0A69
	                                #statWriteReq.data[36] := B#16#10; // Read parameter values
	                                #statWriteReq.data[37] := B#16#01; // Number of elements
	                                #statWriteReq.data[38] := B#16#0A; // Parameter number r2665 (setpoint position) high byte
	                                #statWriteReq.data[39] := B#16#69; // Parameter number r2665 (setpoint position) low byte
	                                #statWriteReq.data[40] := B#16#00; // Subindex
	                                #statWriteReq.data[41] := B#16#00; // Subindex
	                                // 8. Drive parameter r2521[0] (actual position) in hex 0x09D9
	                                #statWriteReq.data[42] := B#16#10; // Read parameter values
	                                #statWriteReq.data[43] := B#16#01; // Number of elements
	                                #statWriteReq.data[44] := B#16#09; // Parameter number r2521[0] (actual position) high byte
	                                #statWriteReq.data[45] := B#16#D9; // Parameter number r2521[0] (actual position) low byte
	                                #statWriteReq.data[46] := B#16#00; // Subindex
	                                #statWriteReq.data[47] := B#16#00; // Subindex
	                                // 9. Drive parameter r2496 (length unit) in hex 0x09C0
	                                #statWriteReq.data[48] := B#16#10; // Read parameter values
	                                #statWriteReq.data[49] := B#16#01; // Number of elements
	                                #statWriteReq.data[50] := B#16#09; // Parameter number r2496 (length unit) high byte
	                                #statWriteReq.data[51] := B#16#C0; // Parameter number r2496 (length unit) low byte
	                                #statWriteReq.data[52] := B#16#00; // Subindex
	                                #statWriteReq.data[53] := B#16#00; // Subindex
	                                // 10. Drive parameter r2497 (velocity unit) in hex 0x09C1
	                                #statWriteReq.data[54] := B#16#10; // Read parameter values
	                                #statWriteReq.data[55] := B#16#01; // Number of elements
	                                #statWriteReq.data[56] := B#16#09; // Parameter number r2497 (velocity unit) high byte
	                                #statWriteReq.data[57] := B#16#C1; // Parameter number r2497 (velocity unit) low byte
	                                #statWriteReq.data[58] := B#16#00; // Subindex
	                                #statWriteReq.data[59] := B#16#00; // Subindex
	                                // 11. Drive parameter r2682 (residual distance) in hex 0x0A7A
	                                #statWriteReq.data[60] := B#16#10; // Read parameter values
	                                #statWriteReq.data[61] := B#16#01; // Number of elements
	                                #statWriteReq.data[62] := B#16#0A; // Parameter number r2682 (residual distance) high byte
	                                #statWriteReq.data[63] := B#16#7A; // Parameter number r2682 (residual distance) low byte
	                                #statWriteReq.data[64] := B#16#00; // Subindex
	                                #statWriteReq.data[65] := B#16#00; // Subindex
	                                // 12. Drive parameter r2565 (following error) in hex 0x0A05
	                                #statWriteReq.data[66] := B#16#10; // Read parameter values
	                                #statWriteReq.data[67] := B#16#01; // Number of elements
	                                #statWriteReq.data[68] := B#16#0A; // Parameter number r2565 (following error) high byte
	                                #statWriteReq.data[69] := B#16#05; // Parameter number r2565 (following error) low byte
	                                #statWriteReq.data[70] := B#16#00; // Subindex
	                                #statWriteReq.data[71] := B#16#00; // Subindex
	                                // 13. Drive parameter r2050[1] (positioning control word) in hex 0x0802
	                                #statWriteReq.data[72] := B#16#10; // Read parameter values
	                                #statWriteReq.data[73] := B#16#01; // Number of elements
	                                #statWriteReq.data[74] := B#16#08; // Parameter number r2050[1] (positioning control word) high byte
	                                #statWriteReq.data[75] := B#16#02; // Parameter number r2050[1] (positioning control word) low byte
	                                #statWriteReq.data[76] := B#16#00; // Subindex
	                                #statWriteReq.data[77] := B#16#01; // Subindex
	                                // 14. Drive parameter c2053[1] (positioning status word) in hex 0x0805
	                                #statWriteReq.data[78] := B#16#10; // Read parameter values
	                                #statWriteReq.data[79] := B#16#01; // Number of elements
	                                #statWriteReq.data[80] := B#16#08; // Parameter number c2053[1] (positioning status word) high byte
	                                #statWriteReq.data[81] := B#16#05; // Parameter number c2053[1] (positioning status word) low byte
	                                #statWriteReq.data[82] := B#16#00; // Subindex
	                                #statWriteReq.data[83] := B#16#01; // Subindex
	                                // 15. Drive parameter c2642 (MDI setpoint position) in hex 0x0A52
	                                #statWriteReq.data[84] := B#16#10; // Read parameter values
	                                #statWriteReq.data[85] := B#16#01; // Number of elements
	                                #statWriteReq.data[86] := B#16#0A; // Parameter number c2642 (MDI setpoint position) high byte
	                                #statWriteReq.data[87] := B#16#52; // Parameter number c2642 (MDI setpoint position) low byte
	                                #statWriteReq.data[88] := B#16#00; // Subindex
	                                #statWriteReq.data[89] := B#16#00; // Subindex
	                                // 16. Drive parameter c2053[0] (#status word) in hex 0x0805
	                                #statWriteReq.data[90] := B#16#10; // Read parameter values
	                                #statWriteReq.data[91] := B#16#01; // Number of elements
	                                #statWriteReq.data[92] := B#16#08; // Parameter number c2053 (status word) high byte
	                                #statWriteReq.data[93] := B#16#05; // Parameter number c2053 (status word) low byte
	                                #statWriteReq.data[94] := B#16#00; // Subindex
	                                #statWriteReq.data[95] := B#16#00; // Subindex
	                                // Start request
	                                #statWriteReqSet := TRUE;
	                                #statDataTransRun := TRUE;
	                            END_REGION S210

	                        ELSE
	                            REGION ELSE
	                                // Type of SINAMICS not found --> delete interface
	                                #tempReferenceDesignator := WSTRING#'';
	                                #moduleInterface.sina.sinaType := 0;
	                                #moduleInterface.sina.statusWord := W#16#0;
	                                #moduleInterface.sina.eposStatusWord1 := W#16#0;
	                                #moduleInterface.sina.eposStatusWord2 := W#16#0;
	                                #moduleInterface.sina.operatingDisplay := 0;
	                                #moduleInterface.sina.override := 0.0;
	                                #moduleInterface.sina.posSetValue := 0.0;
	                                #moduleInterface.sina.posActValue := 0.0;
	                                #moduleInterface.sina.velSetValue := 0.0;
	                                #moduleInterface.sina.velActValue := 0.0;
	                                #moduleInterface.sina.lengthUnit := 0;
	                                #moduleInterface.sina.velocityUnit := 0;
	                                #moduleInterface.sina.residualDistance := 0.0;
	                                #moduleInterface.sina.followingError := 0.0;
	                                #moduleInterface.sina.posControlWord := W#16#0;
	                                #moduleInterface.sina.posStatusWord := W#16#0;
	                                #moduleInterface.sina.blockSelected := 0;
	                                #moduleInterface.sina.blockActive := 0;
	                                #moduleInterface.sina.mdiPosSetValue := 0.0;
	                            END_REGION ELSE
	                    END_CASE;

	                    // Trigger new write request with 1 sec delay (1 sec delay for first trigger and after error of write/read request)
	                    IF #statWriteReqSet AND (#statActTimerValueAct - #statPrevTimeValue) > T#1s THEN
	                        #instWriteRecord.REQ := TRUE;
	                        #statWriteReqSet := FALSE;
	                        #statPrevTimeValue := #statActTimerValueAct;
	                    END_IF;

	                    // Call timer for write/read requests (3 sec delay between each write request)
	                    #instReqTimer.TON(IN := #instWriteRecord.REQ,
	                                      PT := T#3s,
	                                      Q => #tempReadReqTimerOut,
	                                      ET => #statActTimerValueReq);

	                    // Trigger read request and retrigger write request each 3 sec to get updated data
	                    IF #tempReadReqTimerOut THEN
	                        #instWriteRecord.REQ := FALSE;
	                        #instReadRecord.REQ := TRUE;
	                    END_IF;

	                    // Call write request (WRREC)
	                    #instWriteRecord(ID := #tempSinaHwID,
	                                     INDEX := #DPV1_INDEX_DB47,
	                                     LEN := #DPV1_LENGH_DATA,
	                                     RECORD := #statWriteReq);

	                    // Stop write request after error
	                    IF #instWriteRecord.ERROR AND (#statActTimerValueAct - #statPrevTimeValue) > T#1s THEN
	                        #statDataTransRun := FALSE;
	                        #instWriteRecord.REQ := FALSE;
	                        #statPrevTimeValue := #statActTimerValueAct;
	                    END_IF;

	                    // Save status for debugging
	                    IF #instWriteRecord.ERROR THEN
	                        #statusWriteRecord := #instWriteRecord.STATUS;
	                    END_IF;
	                END_REGION Write request

	                REGION Read request
	                    // Stop read request after valid data response
	                    IF #instReadRecord.VALID AND (#statActTimerValueAct - #statPrevTimeValue) > T#1s THEN
	                        #instReadRecord.REQ := FALSE;
	                        #statPrevTimeValue := #statActTimerValueAct;
	                    END_IF;

	                    // Stop read request after error
	                    IF #instReadRecord.ERROR AND (#statActTimerValueAct - #statPrevTimeValue) > T#1s THEN
	                        #statDataTransRun := FALSE;
	                        #instReadRecord.REQ := FALSE;
	                        #statPrevTimeValue := #statActTimerValueAct;
	                    END_IF;

	                    // Save status for debugging
	                    IF #instReadRecord.ERROR THEN
	                        #statusReadRecord := #instReadRecord.STATUS;
	                    END_IF;

	                    // Call read request (RDREC)
	                    #instReadRecord(ID := #tempSinaHwID,
	                                    INDEX := #DPV1_INDEX_DB47,
	                                    MLEN := #DPV1_LENGH_DATA,
	                                    RECORD := #statReadReq);

	                    // Copy valid data from read response to HMI interface
	                    IF #instReadRecord.VALID AND #statReadReq.header.reqRef <> B#16#0 THEN
	                        // Read response is related to write request via order reference "REQ_REF"
	                        // Order reference from write request is mirrowed in read response
	                        CASE #statReadReq.header.reqRef OF
	                            #REQ_REF_S120:
	                                REGION S120
	                                    // EPOS status word 1
	                                    #moduleInterface.sina.eposStatusWord1.%B1 := #statReadReq.data[2]; // high byte
	                                    #moduleInterface.sina.eposStatusWord1.%B0 := #statReadReq.data[3]; // low byte
	                                    // EPOS status word 2
	                                    #moduleInterface.sina.eposStatusWord2.%B1 := #statReadReq.data[6]; // high byte
	                                    #moduleInterface.sina.eposStatusWord2.%B0 := #statReadReq.data[7]; // low byte
	                                    // Operating display
	                                    #tempValueWord.%B1 := #statReadReq.data[10];
	                                    #tempValueWord.%B0 := #statReadReq.data[11];
	                                    #moduleInterface.sina.operatingDisplay := WORD_TO_UINT(#tempValueWord);
	                                    // Override
	                                    #tempValueDword.%B3 := #statReadReq.data[14];
	                                    #tempValueDword.%B2 := #statReadReq.data[15];
	                                    #tempValueDword.%B1 := #statReadReq.data[16];
	                                    #tempValueDword.%B0 := #statReadReq.data[17];
	                                    #moduleInterface.sina.override := DWORD_TO_REAL(#tempValueDword);
	                                    // Setpoint velocity
	                                    #tempValueDword.%B3 := #statReadReq.data[20];
	                                    #tempValueDword.%B2 := #statReadReq.data[21];
	                                    #tempValueDword.%B1 := #statReadReq.data[22];
	                                    #tempValueDword.%B0 := #statReadReq.data[23];
	                                    #moduleInterface.sina.velSetValue := DINT_TO_REAL(DWORD_TO_DINT(#tempValueDword));
	                                    // Actual velocity
	                                    #tempValueDword.%B3 := #statReadReq.data[26];
	                                    #tempValueDword.%B2 := #statReadReq.data[27];
	                                    #tempValueDword.%B1 := #statReadReq.data[28];
	                                    #tempValueDword.%B0 := #statReadReq.data[29];
	                                    #moduleInterface.sina.velActValue := DINT_TO_REAL(DWORD_TO_DINT(#tempValueDword));
	                                    // Setpoint position
	                                    #tempValueDword.%B3 := #statReadReq.data[32];
	                                    #tempValueDword.%B2 := #statReadReq.data[33];
	                                    #tempValueDword.%B1 := #statReadReq.data[34];
	                                    #tempValueDword.%B0 := #statReadReq.data[35];
	                                    #moduleInterface.sina.posSetValue := DINT_TO_REAL(DWORD_TO_DINT(#tempValueDword));
	                                    // Actual position
	                                    #tempValueDword.%B3 := #statReadReq.data[38];
	                                    #tempValueDword.%B2 := #statReadReq.data[39];
	                                    #tempValueDword.%B1 := #statReadReq.data[40];
	                                    #tempValueDword.%B0 := #statReadReq.data[41];
	                                    #moduleInterface.sina.posActValue := DINT_TO_REAL(DWORD_TO_DINT(#tempValueDword));
	                                    // Length unit
	                                    #moduleInterface.sina.lengthUnit := 0; // Only LUs supported
	                                    // Velocity unit
	                                    #moduleInterface.sina.velocityUnit := 0; // Only 1000LU/min supported
	                                    // Residual distance
	                                    #tempValueDword.%B3 := #statReadReq.data[44];
	                                    #tempValueDword.%B2 := #statReadReq.data[45];
	                                    #tempValueDword.%B1 := #statReadReq.data[46];
	                                    #tempValueDword.%B0 := #statReadReq.data[47];
	                                    #moduleInterface.sina.residualDistance := DINT_TO_REAL(DWORD_TO_DINT(#tempValueDword));
	                                    // Following error
	                                    #tempValueDword.%B3 := #statReadReq.data[50];
	                                    #tempValueDword.%B2 := #statReadReq.data[51];
	                                    #tempValueDword.%B1 := #statReadReq.data[52];
	                                    #tempValueDword.%B0 := #statReadReq.data[53];
	                                    #moduleInterface.sina.followingError := DINT_TO_REAL(DWORD_TO_DINT(#tempValueDword));
	                                    // Positioning control word
	                                    #moduleInterface.sina.posControlWord.%B1 := #statReadReq.data[56]; // high byte
	                                    #moduleInterface.sina.posControlWord.%B0 := #statReadReq.data[57]; // low byte
	                                    // Positioning status word
	                                    #moduleInterface.sina.posStatusWord.%B1 := #statReadReq.data[60]; // high byte
	                                    #moduleInterface.sina.posStatusWord.%B0 := #statReadReq.data[61]; // low byte
	                                    // Selected traversing block
	                                    #moduleInterface.sina.blockSelected.%X0 := #moduleInterface.sina.posControlWord.%X0;
	                                    #moduleInterface.sina.blockSelected.%X1 := #moduleInterface.sina.posControlWord.%X1;
	                                    #moduleInterface.sina.blockSelected.%X2 := #moduleInterface.sina.posControlWord.%X2;
	                                    #moduleInterface.sina.blockSelected.%X3 := #moduleInterface.sina.posControlWord.%X3;
	                                    #moduleInterface.sina.blockSelected.%X4 := #moduleInterface.sina.posControlWord.%X4;
	                                    #moduleInterface.sina.blockSelected.%X5 := #moduleInterface.sina.posControlWord.%X5;
	                                    // Active traversing block
	                                    #moduleInterface.sina.blockActive.%X0 := #moduleInterface.sina.posStatusWord.%X0;
	                                    #moduleInterface.sina.blockActive.%X1 := #moduleInterface.sina.posStatusWord.%X1;
	                                    #moduleInterface.sina.blockActive.%X2 := #moduleInterface.sina.posStatusWord.%X2;
	                                    #moduleInterface.sina.blockActive.%X3 := #moduleInterface.sina.posStatusWord.%X3;
	                                    #moduleInterface.sina.blockActive.%X4 := #moduleInterface.sina.posStatusWord.%X4;
	                                    #moduleInterface.sina.blockActive.%X5 := #moduleInterface.sina.posStatusWord.%X5;
	                                    // MID setpoint position
	                                    #tempValueDword.%B3 := #statReadReq.data[64];
	                                    #tempValueDword.%B2 := #statReadReq.data[65];
	                                    #tempValueDword.%B1 := #statReadReq.data[66];
	                                    #tempValueDword.%B0 := #statReadReq.data[67];
	                                    #moduleInterface.sina.mdiPosSetValue := DINT_TO_REAL(DWORD_TO_DINT(#tempValueDword));
	                                    // Status word
	                                    #moduleInterface.sina.statusWord.%B1 := #statReadReq.data[70]; // high byte
	                                    #moduleInterface.sina.statusWord.%B0 := #statReadReq.data[71]; // low byte
	                                END_REGION S120

	                            #REQ_REF_S200:
	                                REGION S200
	                                    // EPOS status word 1
	                                    #moduleInterface.sina.eposStatusWord1.%B1 := #statReadReq.data[2]; // high byte
	                                    #moduleInterface.sina.eposStatusWord1.%B0 := #statReadReq.data[3]; // low byte
	                                    // EPOS status word 2
	                                    #moduleInterface.sina.eposStatusWord2.%B1 := #statReadReq.data[6]; // high byte
	                                    #moduleInterface.sina.eposStatusWord2.%B0 := #statReadReq.data[7]; // low byte
	                                    // Operating display
	                                    #tempValueWord.%B1 := #statReadReq.data[10];
	                                    #tempValueWord.%B0 := #statReadReq.data[11];
	                                    #moduleInterface.sina.operatingDisplay := WORD_TO_UINT(#tempValueWord);
	                                    // Override
	                                    #tempValueDword.%B3 := #statReadReq.data[14];
	                                    #tempValueDword.%B2 := #statReadReq.data[15];
	                                    #tempValueDword.%B1 := #statReadReq.data[16];
	                                    #tempValueDword.%B0 := #statReadReq.data[17];
	                                    #moduleInterface.sina.override := DWORD_TO_REAL(#tempValueDword);
	                                    // Setpoint velocity
	                                    #tempValueDword.%B3 := #statReadReq.data[20];
	                                    #tempValueDword.%B2 := #statReadReq.data[21];
	                                    #tempValueDword.%B1 := #statReadReq.data[22];
	                                    #tempValueDword.%B0 := #statReadReq.data[23];
	                                    #moduleInterface.sina.velSetValue := DWORD_TO_REAL(#tempValueDword);
	                                    // Actual velocity
	                                    #tempValueDword.%B3 := #statReadReq.data[26];
	                                    #tempValueDword.%B2 := #statReadReq.data[27];
	                                    #tempValueDword.%B1 := #statReadReq.data[28];
	                                    #tempValueDword.%B0 := #statReadReq.data[29];
	                                    #moduleInterface.sina.velActValue := DWORD_TO_REAL(#tempValueDword);
	                                    // Setpoint position
	                                    #tempValueDword.%B3 := #statReadReq.data[32];
	                                    #tempValueDword.%B2 := #statReadReq.data[33];
	                                    #tempValueDword.%B1 := #statReadReq.data[34];
	                                    #tempValueDword.%B0 := #statReadReq.data[35];
	                                    #moduleInterface.sina.posSetValue := DWORD_TO_REAL(#tempValueDword);
	                                    // Actual position
	                                    #tempValueDword.%B3 := #statReadReq.data[38];
	                                    #tempValueDword.%B2 := #statReadReq.data[39];
	                                    #tempValueDword.%B1 := #statReadReq.data[40];
	                                    #tempValueDword.%B0 := #statReadReq.data[41];
	                                    #moduleInterface.sina.posActValue := DWORD_TO_REAL(#tempValueDword);
	                                    // Length unit
	                                    #tempValueWord.%B1 := #statReadReq.data[44];
	                                    #tempValueWord.%B0 := #statReadReq.data[45];
	                                    #moduleInterface.sina.lengthUnit := WORD_TO_INT(#tempValueWord);
	                                    // Velocity unit
	                                    #tempValueWord.%B1 := #statReadReq.data[48];
	                                    #tempValueWord.%B0 := #statReadReq.data[49];
	                                    #moduleInterface.sina.velocityUnit := WORD_TO_INT(#tempValueWord);
	                                    // Residual distance
	                                    #tempValueDword.%B3 := #statReadReq.data[52];
	                                    #tempValueDword.%B2 := #statReadReq.data[53];
	                                    #tempValueDword.%B1 := #statReadReq.data[54];
	                                    #tempValueDword.%B0 := #statReadReq.data[55];
	                                    #moduleInterface.sina.residualDistance := DWORD_TO_REAL(#tempValueDword);
	                                    // Following error
	                                    #tempValueDword.%B3 := #statReadReq.data[58];
	                                    #tempValueDword.%B2 := #statReadReq.data[59];
	                                    #tempValueDword.%B1 := #statReadReq.data[60];
	                                    #tempValueDword.%B0 := #statReadReq.data[61];
	                                    #moduleInterface.sina.followingError := DWORD_TO_REAL(#tempValueDword);
	                                    // Positioning control word
	                                    #moduleInterface.sina.posControlWord.%B1 := #statReadReq.data[64]; // high byte
	                                    #moduleInterface.sina.posControlWord.%B0 := #statReadReq.data[65]; // low byte
	                                    // Positioning status word
	                                    #moduleInterface.sina.posStatusWord.%B1 := #statReadReq.data[68]; // high byte
	                                    #moduleInterface.sina.posStatusWord.%B0 := #statReadReq.data[69]; // low byte
	                                    // Selected traversing block
	                                    #moduleInterface.sina.blockSelected.%X0 := #moduleInterface.sina.posControlWord.%X0;
	                                    #moduleInterface.sina.blockSelected.%X1 := #moduleInterface.sina.posControlWord.%X1;
	                                    #moduleInterface.sina.blockSelected.%X2 := #moduleInterface.sina.posControlWord.%X2;
	                                    #moduleInterface.sina.blockSelected.%X3 := #moduleInterface.sina.posControlWord.%X3;
	                                    #moduleInterface.sina.blockSelected.%X4 := #moduleInterface.sina.posControlWord.%X4;
	                                    #moduleInterface.sina.blockSelected.%X5 := #moduleInterface.sina.posControlWord.%X5;
	                                    // Active traversing block
	                                    #moduleInterface.sina.blockActive.%X0 := #moduleInterface.sina.posStatusWord.%X0;
	                                    #moduleInterface.sina.blockActive.%X1 := #moduleInterface.sina.posStatusWord.%X1;
	                                    #moduleInterface.sina.blockActive.%X2 := #moduleInterface.sina.posStatusWord.%X2;
	                                    #moduleInterface.sina.blockActive.%X3 := #moduleInterface.sina.posStatusWord.%X3;
	                                    #moduleInterface.sina.blockActive.%X4 := #moduleInterface.sina.posStatusWord.%X4;
	                                    #moduleInterface.sina.blockActive.%X5 := #moduleInterface.sina.posStatusWord.%X5;
	                                    // MID setpoint position
	                                    #tempValueDword.%B3 := #statReadReq.data[72];
	                                    #tempValueDword.%B2 := #statReadReq.data[73];
	                                    #tempValueDword.%B1 := #statReadReq.data[74];
	                                    #tempValueDword.%B0 := #statReadReq.data[75];
	                                    #moduleInterface.sina.mdiPosSetValue := DWORD_TO_REAL(#tempValueDword);
	                                    // Status word
	                                    #moduleInterface.sina.statusWord.%B1 := #statReadReq.data[78]; // high byte
	                                    #moduleInterface.sina.statusWord.%B0 := #statReadReq.data[79]; // low byte
	                                END_REGION S200

	                            #REQ_REF_S210:
	                                REGION S210
	                                    // EPOS status word 1
	                                    #moduleInterface.sina.eposStatusWord1.%B1 := #statReadReq.data[2]; // high byte
	                                    #moduleInterface.sina.eposStatusWord1.%B0 := #statReadReq.data[3]; // low byte
	                                    // EPOS status word 2
	                                    #moduleInterface.sina.eposStatusWord2.%B1 := #statReadReq.data[6]; // high byte
	                                    #moduleInterface.sina.eposStatusWord2.%B0 := #statReadReq.data[7]; // low byte
	                                    // Operating display
	                                    #tempValueWord.%B1 := #statReadReq.data[10];
	                                    #tempValueWord.%B0 := #statReadReq.data[11];
	                                    #moduleInterface.sina.operatingDisplay := WORD_TO_UINT(#tempValueWord);
	                                    // Override
	                                    #tempValueDword.%B3 := #statReadReq.data[14];
	                                    #tempValueDword.%B2 := #statReadReq.data[15];
	                                    #tempValueDword.%B1 := #statReadReq.data[16];
	                                    #tempValueDword.%B0 := #statReadReq.data[17];
	                                    #moduleInterface.sina.override := DWORD_TO_REAL(#tempValueDword);
	                                    // Setpoint velocity
	                                    #tempValueDword.%B3 := #statReadReq.data[20];
	                                    #tempValueDword.%B2 := #statReadReq.data[21];
	                                    #tempValueDword.%B1 := #statReadReq.data[22];
	                                    #tempValueDword.%B0 := #statReadReq.data[23];
	                                    #moduleInterface.sina.velSetValue := DWORD_TO_REAL(#tempValueDword);
	                                    // Actual velocity
	                                    #tempValueDword.%B3 := #statReadReq.data[26];
	                                    #tempValueDword.%B2 := #statReadReq.data[27];
	                                    #tempValueDword.%B1 := #statReadReq.data[28];
	                                    #tempValueDword.%B0 := #statReadReq.data[29];
	                                    #moduleInterface.sina.velActValue := DWORD_TO_REAL(#tempValueDword);
	                                    // Setpoint position
	                                    #tempValueDword.%B3 := #statReadReq.data[32];
	                                    #tempValueDword.%B2 := #statReadReq.data[33];
	                                    #tempValueDword.%B1 := #statReadReq.data[34];
	                                    #tempValueDword.%B0 := #statReadReq.data[35];
	                                    #moduleInterface.sina.posSetValue := DWORD_TO_REAL(#tempValueDword);
	                                    // Actual position
	                                    #tempValueDword.%B3 := #statReadReq.data[38];
	                                    #tempValueDword.%B2 := #statReadReq.data[39];
	                                    #tempValueDword.%B1 := #statReadReq.data[40];
	                                    #tempValueDword.%B0 := #statReadReq.data[41];
	                                    #moduleInterface.sina.posActValue := DWORD_TO_REAL(#tempValueDword);
	                                    // Length unit
	                                    #tempValueWord.%B1 := #statReadReq.data[44];
	                                    #tempValueWord.%B0 := #statReadReq.data[45];
	                                    #moduleInterface.sina.lengthUnit := WORD_TO_INT(#tempValueWord);
	                                    // Velocity unit
	                                    #tempValueWord.%B1 := #statReadReq.data[48];
	                                    #tempValueWord.%B0 := #statReadReq.data[49];
	                                    #moduleInterface.sina.velocityUnit := WORD_TO_INT(#tempValueWord);
	                                    // Residual distance
	                                    #tempValueDword.%B3 := #statReadReq.data[52];
	                                    #tempValueDword.%B2 := #statReadReq.data[53];
	                                    #tempValueDword.%B1 := #statReadReq.data[54];
	                                    #tempValueDword.%B0 := #statReadReq.data[55];
	                                    #moduleInterface.sina.residualDistance := DWORD_TO_REAL(#tempValueDword);
	                                    // Following error
	                                    #tempValueDword.%B3 := #statReadReq.data[58];
	                                    #tempValueDword.%B2 := #statReadReq.data[59];
	                                    #tempValueDword.%B1 := #statReadReq.data[60];
	                                    #tempValueDword.%B0 := #statReadReq.data[61];
	                                    #moduleInterface.sina.followingError := DWORD_TO_REAL(#tempValueDword);
	                                    // Positioning control word
	                                    #moduleInterface.sina.posControlWord.%B1 := #statReadReq.data[64]; // high byte
	                                    #moduleInterface.sina.posControlWord.%B0 := #statReadReq.data[65]; // low byte
	                                    // Positioning status word
	                                    #moduleInterface.sina.posStatusWord.%B1 := #statReadReq.data[68]; // high byte
	                                    #moduleInterface.sina.posStatusWord.%B0 := #statReadReq.data[69]; // low byte
	                                    // Selected traversing block
	                                    #moduleInterface.sina.blockSelected.%X0 := #moduleInterface.sina.posControlWord.%X0;
	                                    #moduleInterface.sina.blockSelected.%X1 := #moduleInterface.sina.posControlWord.%X1;
	                                    #moduleInterface.sina.blockSelected.%X2 := #moduleInterface.sina.posControlWord.%X2;
	                                    #moduleInterface.sina.blockSelected.%X3 := #moduleInterface.sina.posControlWord.%X3;
	                                    #moduleInterface.sina.blockSelected.%X4 := #moduleInterface.sina.posControlWord.%X4;
	                                    #moduleInterface.sina.blockSelected.%X5 := #moduleInterface.sina.posControlWord.%X5;
	                                    // Active traversing block
	                                    #moduleInterface.sina.blockActive.%X0 := #moduleInterface.sina.posStatusWord.%X0;
	                                    #moduleInterface.sina.blockActive.%X1 := #moduleInterface.sina.posStatusWord.%X1;
	                                    #moduleInterface.sina.blockActive.%X2 := #moduleInterface.sina.posStatusWord.%X2;
	                                    #moduleInterface.sina.blockActive.%X3 := #moduleInterface.sina.posStatusWord.%X3;
	                                    #moduleInterface.sina.blockActive.%X4 := #moduleInterface.sina.posStatusWord.%X4;
	                                    #moduleInterface.sina.blockActive.%X5 := #moduleInterface.sina.posStatusWord.%X5;
	                                    // MID setpoint position
	                                    #tempValueDword.%B3 := #statReadReq.data[72];
	                                    #tempValueDword.%B2 := #statReadReq.data[73];
	                                    #tempValueDword.%B1 := #statReadReq.data[74];
	                                    #tempValueDword.%B0 := #statReadReq.data[75];
	                                    #moduleInterface.sina.mdiPosSetValue := DWORD_TO_REAL(#tempValueDword);
	                                    // Status word
	                                    #moduleInterface.sina.statusWord.%B1 := #statReadReq.data[78]; // high byte
	                                    #moduleInterface.sina.statusWord.%B0 := #statReadReq.data[79]; // low byte
	                                END_REGION S210
	                        END_CASE;
	                    END_IF;
	                END_REGION Read request
	            END_REGION Processing

	        #FB_STATE_DISABLING: // Disabling active
	            REGION Disabling
	                // Delete interface
	                #statusWriteRecord := W#16#00;
	                #statusReadRecord := W#16#00;
	                #statPrevDriveIndex := #DRV_INDEX_INIT;
	                #tempReferenceDesignator := WSTRING#'';
	                #moduleInterface.sina.sinaType := 0;
	                #moduleInterface.sina.statusWord := W#16#0;
	                #moduleInterface.sina.eposStatusWord1 := W#16#0;
	                #moduleInterface.sina.eposStatusWord2 := W#16#0;
	                #moduleInterface.sina.operatingDisplay := 0;
	                #moduleInterface.sina.override := 0.0;
	                #moduleInterface.sina.posSetValue := 0.0;
	                #moduleInterface.sina.posActValue := 0.0;
	                #moduleInterface.sina.velSetValue := 0.0;
	                #moduleInterface.sina.velActValue := 0.0;
	                #moduleInterface.sina.lengthUnit := 0;
	                #moduleInterface.sina.velocityUnit := 0;
	                #moduleInterface.sina.residualDistance := 0.0;
	                #moduleInterface.sina.followingError := 0.0;
	                #moduleInterface.sina.posControlWord := W#16#0;
	                #moduleInterface.sina.posStatusWord := W#16#0;
	                #moduleInterface.sina.blockSelected := 0;
	                #moduleInterface.sina.blockActive := 0;
	                #moduleInterface.sina.mdiPosSetValue := 0.0;
	                // When disabling is complete the '#statDisablingCompleted' must be set
	                #statInternal.disablingCompleted := TRUE;
	            END_REGION Disabling

	        ELSE // Undefined state in state machine reached
	            REGION Undefined state
	                #statInternal.diagnostics.status := #ERR_UNDEFINED_STATE;
	                #statInternal.diagnostics.subfunctionStatus := #SUB_STATUS_NO_ERROR;
	                #statInternal.diagnostics.stateNumber := #statMainState;
	                #statInternal.errorUserCleared := TRUE;
	            END_REGION Undefined state
	    END_CASE;
	END_REGION STATE MACHINE

	REGION OUTPUTS
	    // Write outputs
	    IF (#statInternal.disablingCompleted = TRUE) THEN
	        REGION Disabling
	            // Reset outputs if disabling completed
	            #statInternal.valid := FALSE;
	            #statInternal.busy := FALSE;
	            #statInternal.error := FALSE;
	            #statInternal.errorUserCleared := FALSE;
	            #statInternal.errorAutoCleared := FALSE;
	            #statInternal.diagnostics.status := #STATUS_NO_CALL;
	            #statMainState := #FB_STATE_NO_PROCESSING;
	        END_REGION Disabling

	    ELSIF (#statInternal.errorUserCleared = TRUE) AND (#statInternal.error = FALSE) THEN
	        REGION Error user cleared
	            // Error can only be cleared by user; rising edge for 'tempEnable' is needed to continue
	            #statInternal.valid := FALSE;
	            #statInternal.busy := FALSE;
	            #statInternal.error := TRUE;
	            // Write diagnostics
	            //#diagnostics := #statDiagnostic;
	            #diagnostics := #statInternal.diagnostics;
	            // execution aborted --> set state no processing
	            #statMainState := #FB_STATE_NO_PROCESSING;
	        END_REGION Error user cleared

	    ELSIF (#statInternal.errorAutoCleared = TRUE) AND (#statInternal.error = FALSE) THEN
	        REGION Error auto cleared
	            // Error can be reset by FB automatically
	            #statInternal.valid := FALSE;
	            #statInternal.busy := TRUE;
	            #statInternal.error := TRUE;
	            // Write diagnostics
	            #diagnostics := #statInternal.diagnostics;
	        END_REGION Error auto cleared

	    ELSIF (#statInternal.errorAutoCleared = FALSE) AND (#statInternal.errorUserCleared = FALSE) AND (#statInternal.error = TRUE) THEN
	        REGION After user/auto cleared or command aborted
	            // If autocleared error is acknowledged
	            #statInternal.valid := TRUE;
	            #statInternal.busy := TRUE;
	            #statInternal.error := FALSE;
	        END_REGION After user/auto cleared or command aborted
	    END_IF;

	    REGION Write static/temp values to outputs
	        #valid := #statInternal.valid;
	        #busy := #statInternal.busy;
	        #error := #statInternal.error;
	        #status := #statInternal.diagnostics.status;
	        // ENO mechanism
	        ENO := NOT #statInternal.error;
	        // Application specific values to outputs
	        #moduleInterface.hmi.referenceDesignator := #tempReferenceDesignator;
	    END_REGION Write static/temp values to outputs
	END_REGION OUTPUTS

END_FUNCTION_BLOCK

